{attribute addProperty BoxType "EK1100-0000-0018"}
{attribute addProperty Id "Beckhoff_CXxxxxEK1122Beckhoff_CXxxxxEK1122_73DAF5DE4544568"}
{attribute addProperty CRC "1360403376"}
{attribute addProperty SizeInBites "4544"}
{attribute addProperty SizeInBytes "568"}
TYPE Beckhoff_CXxxxx_51161BB0 EXTENDS EK1100_179A0949 :
STRUCT
	{attribute addProperty Name "Beckhoff_CXxxxxEK1122"}
	Beckhoff_CXxxxxEK1122 : Beckhoff_CXxxxxEK1122_73DAF5DE;
END_STRUCT
END_TYPE

(* stored: Version 1.2.0.0, ProductVersion 3.1.4024.9
   DUT Beckhoff_CXxxxx_51161BB0: Id {4113e3a3-6358-424c-8c3c-5bd4a16363b2} *)
